Staubli VAL3: save.pgx

public program save(num& x_nResult[])
begin
  x_nResult=saveInOut:libSave()
  if x_nResult!=0
    delay(0.5)
    x_nResult=saveInOut:libSave()
  endIf
end
